(* IEC 61131-3 sources: programs/VI-54/VI-54_20171205/VI-54_20171205/Stations/PLC_VI54/VI-54_171014/Class/_VaranDriveBase (part 2) *)

		s_DataObjectA1.p_Handle^.ucCtrlStat := VARAN_DO_SINGLE_RUN;
	end_if;

	//is Axis 2 in use
	if ( ud_Axis.2 ) then
		s_Axis2Data.e_AxisState := _NoInit;
	else
		s_Axis2Data.e_AxisState := _NotUsed;
//		Axis2_Enable.write( 0 );
//		Axis2_ControlWord.DriveEnable := FALSE;

//		s_Axis2Data.s_WriteValues.a_SyncValues[ 0 ] := ( ( Axis2_ControlWord$DINT shl 16 ) or ( Axis2_SetCurrent and 16#FFFF ) )$DINT;
		s_DataObjectA2.p_DataWrite^.sd_Value1 := s_Axis2Data.s_WriteValues.a_SyncValues[ 0 ];

		s_DataObjectA2.p_Handle^.ucCtrlStat := VARAN_DO_SINGLE_RUN;
	end_if;

	//is Axis 3 in use
	if ( ud_Axis.3 ) then
		s_Axis3Data.e_AxisState := _NoInit;
	else
		s_Axis3Data.e_AxisState := _NotUsed;
//		Axis3_Enable.write( 0 );
//		Axis3_ControlWord.DriveEnable := FALSE;

//		s_Axis3Data.s_WriteValues.a_SyncValues[ 0 ] := ( ( Axis3_ControlWord$DINT shl 16 ) or ( Axis3_SetCurrent and 16#FFFF ) )$DINT;
		s_DataObjectA3.p_DataWrite^.sd_Value1 := s_Axis3Data.s_WriteValues.a_SyncValues[ 0 ];

		s_DataObjectA3.p_Handle^.ucCtrlStat := VARAN_DO_SINGLE_RUN;
	end_if;
*)

(*
	b_InitOk := TRUE;

	InitDrive();
*)
END_FUNCTION

FUNCTION VIRTUAL GLOBAL _VaranDriveBase::State::NewInst
	VAR_INPUT
		pPara 	: ^CmdStruct;
		pResult 	: ^results;
	END_VAR
	VAR_OUTPUT
		ret_code 	: iprStates;
	END_VAR
  VAR
  	pStr_HWTRequested : ^CHAR;
    us_HWTRequestedCurrIndex : USINT;
  END_VAR

  pStr_HWTRequested := NIL;
  us_HWTRequestedCurrIndex := 0;

  ret_code:= READY;

	case ( pPara^.uiCmd ) of
		0 : SetAxisOn( pPara^.aPara[ 0 ]$BDINT );

    1 : // list with parameternumbers to skip

        // check if index in range (0-7)
        //if (pPara^.aPara[2] >= 0) & (pPara^.aPara[2] <= (AxisAvailableNo-1)) then
        if (pPara^.aPara[2] < DIASDRIVE_MAX_AXIS) & (aAxisData[pPara^.aPara[2]].e_AxisState <> _NotUsed) then
          s_SkipParameter[pPara^.aPara[2]].us_No    := to_usint(pPara^.aPara[1]); // number of values in memory
          s_SkipParameter[pPara^.aPara[2]].p_Values := (pPara^.aPara[0])$^USINT; // pointer on memory
        end_if;

    CMD_GET_HARDWARE_DIAGNOSIS :

        ret_code := ERROR;
        pStr_HWTRequested := pPara^.aPara[0]$t_HWCGetHardwareTreeEntryIn.pStr_LastHardewareTreeEntry;

        if pStr_HWTRequested & p_ObjectPath then
          // Needed as default for
          ret_code := READY;

          if (pStr_HWTRequested$^USINT^ = p_ObjectPath^) then // Check if the call was to the Mng
            // Call base 1st as it as info from SPI accesses
            ret_code := Varan_Base::State.NewInst(pPara, pResult);  // Pass on command to base
          end_if;

          if (p_DriveMngBase) then

            // Call Mng, may overwrite some data, has got at least additional info on the FW version
            ret_code := p_DriveMngBase$^VirtualBase^.NewInst(pPara,pResult);

          end_if;
        end_if;

    CMD_GET_HARDWARE_TREE_ENTRY :

        ret_code := ERROR;

        pStr_HWTRequested := pPara^.aPara[0]$t_HWCGetHardwareTreeEntryIn.pStr_LastHardewareTreeEntry;

        // Check HWT String
        if pStr_HWTRequested & p_ObjectPath then

          // Check if the passed string is smaller than the own string
          if pStr_HWTRequested$^USINT^ < p_ObjectPath^ then

            // Call base
            ret_code := Varan_Base::State.NewInst(pPara, pResult);  // Pass on command to base

          // Check if last call was to Base itself
          // Compare string content
          elsif _memcmp( ptr1 := pStr_HWTRequested + 2,
                         ptr2 := p_ObjectPath + 1,
                         cntr := p_ObjectPath^) = 0 then

            // Compare string length
            if (pStr_HWTRequested$^USINT^ = p_ObjectPath^) then

              // Last module called was the Drivemng itself, next module is the 1st axis behind the manager
              if (p_DriveMngBase) then

                ret_code := p_DriveMngBase$^VirtualBase^.NewInst(pPara, pResult); // Pass on command to drive manager

              end_if;

            elsif (pStr_HWTRequested$^USINT^ > p_ObjectPath^ + 1) then // Must be at least 2 Bytey larger, ESCAPE Sequence + Place

              // Check escape sequence
              if ( (pStr_HWTRequested + (p_ObjectPath^) + 2 )^ = HWT_ESCAPE_DRIVE) then // First place after manager Itself is escape sequence + 1 for addional length byte
                // Last Module must have been a Axis Module behind the manager
                // Update index
                pPara^.aPara[0]$t_HWCGetHardwareTreeEntryIn.us_current_index  := p_ObjectPath^ + 3; // Second place after manager Itself is place + 1 for addional length byte
                pPara^.aPara[0]$t_HWCGetHardwareTreeEntryIn.us_current_length := pStr_HWTRequested^ - p_ObjectPath^ - 1;

                if (p_DriveMngBase) then

                  ret_code := p_DriveMngBase$^VirtualBase^.NewInst(pPara, pResult); // Pass on command to drive manager

                end_if;

              else // Length not equal and no Escape sequence, = VARAN Module behind CTMS was called 1.st

                ret_code := Varan_Base::State.NewInst(pPara, pResult);  // Pass on command to base
              end_if;

            else  // Requested string length > this string length, _memcmp failed => Last string was from a differet Varan Port

              ret_code := Varan_Base::State.NewInst(pPara, pResult);  // Pass on command to base
            end_if;

          else
            ret_code := Varan_Base::State.NewInst(pPara, pResult);  // Pass on command to base
          end_if;

        else
          // pStr_HWTRequested is probably nil, pass on command to base
          ret_code := Varan_Base::State.NewInst(pPara, pResult);  // Pass on command to base
        end_if;

	  else
      //Pass on command to base
      ret_code := Varan_Base::State.NewInst(pPara:=pPara, pResult:=pResult);
	end_case;

END_FUNCTION

FUNCTION _VaranDriveBase::SkipEntries
	VAR_INPUT
		us_Axis 	: USINT;
		p_Axis 	: ^t_AxisData;
	END_VAR
  VAR
  	i         : UDINT;
    p_ActPara : ^USINT;
    b_ParaOK  : BOOL;
  END_VAR

  // if there are parameters to skip
  if s_SkipParameter[us_Axis].us_No > 0 then
    b_ParaOK := FALSE;

    // as long as the parameter is skipped and we have have still parameters in the list
    while (b_ParaOK = FALSE) & (p_Axis^.ui_ParaListCnt) do
      // set pointer on first value to skip
      p_ActPara := s_SkipParameter[us_Axis].p_Values;

      b_ParaOK := TRUE;

      // for all skip parameters
      for i := 0 to (s_SkipParameter[us_Axis].us_No - 1) do
        // if the actual parameter number is found in the skip parameter list
        if p_ActPara^ = p_Axis^.p_ParaList^.us_number then
          p_Axis^.ui_ParaListCnt 	-= 1;
          p_Axis^.p_ParaList 		  += sizeof( t_ParaList );

          b_ParaOK := FALSE;
          exit;
        end_if;

        p_ActPara += sizeof(USINT);
      end_for;
    end_while;
  end_if;

END_FUNCTION

FUNCTION GLOBAL _VaranDriveBase::StartCommunication
	VAR_INPUT
		AxisExtend 	: BDINT;
		AxisFast 	: BDINT;
		pServer4CallBack 	: ^BDINT;
	END_VAR

  ExtendedAxisSettings := AxisExtend;
  FastAxisSettings := AxisFast;

  pCallBackServer := pServer4CallBack - sizeof(SvrCh.pMeth);

END_FUNCTION

FUNCTION GLOBAL _VaranDriveBase::GetAxisRdPtr
	VAR_INPUT
		AxisNr 	: DINT;
	END_VAR
	VAR_OUTPUT
		pReadPara 	: ^t_ReadValuePtr;
	END_VAR

  pReadPara := NIL;

  //look which Axis we have
//  if (AxisNr >= 0) & (AxisNr <= (AxisAvailableNo-1)) then
  if (AxisNr < DIASDRIVE_MAX_AXIS) & (aAxisData[AxisNr].e_AxisState <> _NotUsed) then
    pReadPara := #aAxisData[AxisNr].s_ReadValues;
  end_if;

END_FUNCTION

FUNCTION GLOBAL _VaranDriveBase::GetAxisWrPtr
	VAR_INPUT
		AxisNr 	: DINT;
	END_VAR
	VAR_OUTPUT
		pWritePara 	: ^t_WriteValuePtr;
	END_VAR

  pWritePara := NIL;

  //look which Axis we have
//  if (AxisNr >= 0) & (AxisNr <= (AxisAvailableNo-1)) then
  if (AxisNr < DIASDRIVE_MAX_AXIS) & (aAxisData[AxisNr].e_AxisState <> _NotUsed) then
    pWritePara := #aAxisData[AxisNr].s_WriteValues;
  end_if;

END_FUNCTION

FUNCTION GLOBAL _VaranDriveBase::GetDriveIntState
	VAR_OUTPUT
		retcode 	: DINT;
	END_VAR

  // to get the actual state of the rtwork state machine
  // retcode = 3 means Operational (MOD 4 is for model SDD100/5000 to have the same returncodes)
  retcode := e_RtSSW$DINT MOD 4;

END_FUNCTION

FUNCTION _VaranDriveBase::GetObjectValueNew
	VAR_INPUT
		us_Axis 	: USINT;
	END_VAR
  VAR
    p_Axis			: ^t_AxisData;
    p_Write     : ^t_newASYWrite;
    p_Read      : ^t_newASYRead;
  END_VAR

	//------------------------------------------------------------------------------------------------
	//look which Axis we have and set pointers
//  if (us_Axis >= 0) & (us_Axis <= (AxisAvailableNo-1)) then
  if (us_Axis < DIASDRIVE_MAX_AXIS) & (aAxisData[us_Axis].e_AxisState <> _NotUsed) then
    p_Axis	:= #aAxisData[us_Axis];
    p_Read 	:= newAsyDO.p_DataRead + us_Axis * sizeof(t_newASYRead);
    p_Write	:= newAsyDO.p_DataWrite + us_Axis * sizeof(t_newASYWrite);
  else
    //else do nothing (should not come her)
    return;
  end_if;

	//------------------------------------------------------------------------------------------------
	//get to right step
	case ( p_Axis^.us_ParaReady ) of

		_SendExecution: // we wait 1 cycle to ensure that the request is written to the Drive (what object number we want to read or write)
							p_Axis^.us_ParaReady := _ResetExecution;

    _ResetExecution:// now toggle the togglebit to start tell the drive, that the data are complete (no chance for byte errors in this way)

              //send transmit execution request for object handling
							p_Axis^.b_OldToggleState := p_Read^.us_TransmitControl.ToggleBit;

              // toggle toggle bit
              p_Write^.us_DriveControl.ToggleBit := NOT p_Read^.us_TransmitControl.ToggleBit;

							//reset error and go to next step
							p_Axis^.sd_ObjectError := 0;
							p_Axis^.us_ParaReady := _Wait4Response;

		_Wait4Response:		//wait until receive state is true
							if ( p_Read^.us_TransmitControl.ToggleBit <> p_Axis^.b_OldToggleState) then

								//look if we have a parameter list
								if ( p_Axis^.b_ListActive = TRUE ) then

                  // skip all defined parameter entries
                  SkipEntries(us_Axis, p_Axis);

									//have we set all parameter
									if ( p_Axis^.ui_ParaListCnt ) then

										//set data to object handling registers
										p_Write^.us_ObjectAddress					        := p_Axis^.p_ParaList^.us_number;
										p_Write^.sd_ObjectValue					          := p_Axis^.p_ParaList^.sd_value;
										p_Write^.us_DriveControl.ReadWriteObject	:= TRUE;

										//set next parameter step and set pointer to next parameter data
										p_Axis^.us_ParaReady 	:= _SendExecution;
										p_Axis^.ui_ParaListCnt 	-= 1;
										p_Axis^.p_ParaList 		+= sizeof( t_ParaList );

									else
										//set ssw to idle and deactivate parameter list
										p_Axis^.b_ListActive 	:= FALSE;

										//look if we get a parameter list
										if ( p_Axis^.e_AxisState = _NoParaList ) then
											p_Axis^.e_AxisState		:= _NotSynchron;
										end_if;

										p_Axis^.us_ParaReady 	:= _IdleState;

									end_if;

								else
									//get to idle step
									p_Axis^.us_ParaReady := _IdleState;

									//look for an object error
									if ( p_Read^.us_TransmitControl.ErrorInObjectHandling = TRUE ) then
										p_Axis^.sd_ObjectError := p_Read^.sd_ObjectValue;
									else
                 		p_Axis^.sd_Asyncdata := p_Read^.sd_ObjectValue;
                  end_if;

								end_if;
							end_if;

		_IdleState:				//do nothing in this step

	end_case;

END_FUNCTION

FUNCTION _VaranDriveBase::InitAxisNew
	VAR_INPUT
		us_AxisNo 	: USINT;
	END_VAR
	VAR_OUTPUT
		sd_retval 	: DINT;
	END_VAR
  VAR
    p_Axis			: ^t_AxisData;
    p_Write     : ^t_newASYWrite;
    p_Read      : ^t_newASYRead;
    p_data_object : ^t_newISODO;
  END_VAR

	//we do this only if class is not initialized
	if ( State <> _NotInitialized ) then
		return;
	end_if;

	//------------------------------------------------------------------------------------------------
	//look which Axis we have and set pointers
//  if (us_AxisNo >= 0) & (us_AxisNo <= (AxisAvailableNo-1)) then
  if (us_AxisNo < DIASDRIVE_MAX_AXIS) & (aAxisData[us_AxisNo].e_AxisState <> _NotUsed) then
    p_Axis			:= #aAxisData[us_AxisNo];
    p_data_object	:= #newIsoDOs[us_AxisNo];
    p_Read 	:= newAsyDO.p_DataRead + us_AxisNo * sizeof(t_newASYRead);
    p_Write	:= newAsyDO.p_DataWrite + us_AxisNo * sizeof(t_newASYWrite);
  else
    sd_retval := -2;
    return;
  end_if;

	//------------------------------------------------------------------------------------------------
	//look which case we have
	case ( e_InitSSW ) of

		//-----------------------------------------------------------------------------------------------
		_SetDataObjectOn:
					//is Axis in use
					if ( p_Axis^.e_AxisState <> _NotUsed ) then

//Revision 1.20 start
            _memset(p_data_object^.p_DataWrite, 16#00, p_Axis^.ud_DOLength); // reinit the memory before sending
//Revision 1.20 end

						//reset data object of Axis
            if b_PayloadSupport then
              if bAddDOsToListSupport then
                sd_retval := MULTI_VARAN_IINSERTDOINTODOL(p_data_object^.p_Handle$UDINT);
              end_if;
              EnableDO(ud_DOHandle:=p_data_object^.p_Handle$UDINT);
            else
                // Payload DOs automatically use the client Timebase to set the Prescaler of the DOs
              //set right multiplier
              p_data_object^.p_Handle^.ucExePrescaler := VaranTimeMultiplier$USINT - 1;

              ResetDataObject	( p_handleDO	:= p_data_object^.p_Handle
                              , us_state		:= VARAN_DO_CONT_RUN
                                , ud_bytes		:= p_Axis^.ud_DOLength * 2);
            end_if;
(*
            if ( us_AxisNo = 3 & UseFastAxis ) then

              ResetDataObject	( p_handleDO	:= s_DataFastAxis.p_Handle
                              , us_state		:= VARAN_DO_CONT_RUN
                              , ud_bytes		:= sizeof( t_FastAxisRead ) + sizeof( t_FastAxisWrite )
                              );

              s_DataFastAxis.p_DataWrite^.us_TransmittExecution.EnableType2 := TRUE;
            end_if;
*)
						//next step
						e_InitSSW := _SetInitAxis;

					else
						//go to idle state
						e_InitSSW := _CyIdle;
					end_if;

		//-----------------------------------------------------------------------------------------------
		_SetInitAxis:
					//InitAxis
					if ( p_Axis^.e_AxisState = _NoInit ) then

						p_Write^.us_DriveControl.InitCommunication 			:= TRUE;

					end_if;

          p_Axis^.b_OldToggleState := p_Read^.us_TransmitControl.ToggleBit;

          // toggle toggle bit
          p_Write^.us_DriveControl.ToggleBit := NOT p_Read^.us_TransmitControl.ToggleBit;

					//next step and timestamp
					e_InitSSW 		:= _WaitInit;
					ud_TimemarkInit := ops.tAbsolute;

		//-----------------------------------------------------------------------------------------------
		_WaitInit:	//reset startobjecttransfer bit

					//look if Axis 1 must be init
					if ( p_Axis^.e_AxisState = _NoInit ) then

						//object must be executed, error in object handling must be set and error code must be 9
						if (( p_Read^.us_TransmitControl.ToggleBit <> p_Axis^.b_OldToggleState)
                & p_Read^.us_TransmitControl.ErrorInObjectHandling	= TRUE
                & p_Read^.sd_ObjectValue 							= 9
                )
						then
							//set Axis to next state
							p_Axis^.e_AxisState := _NoParaList;
							e_InitSSW := _SetFinishInit;

            //after timeout check again
            elsif ( ops.tAbsolute - ud_TimemarkInit > 1sec ) then
              e_InitSSW := _SetInitAxis;
            end_if;

					//after timeout check again
					elsif ( ops.tAbsolute - ud_TimemarkInit > 1sec ) then
						e_InitSSW := _SetInitAxis;
					end_if;

		//-----------------------------------------------------------------------------------------------
		_SetFinishInit:

					//If Axis is in right state
					if ( p_Axis^.e_AxisState = _NoParaList ) then

						p_Write^.us_DriveControl.InitCommunication 			:= FALSE;
					end_if;

          p_Axis^.b_OldToggleState := p_Read^.us_TransmitControl.ToggleBit;

          // toggle toggle bit
          p_Write^.us_DriveControl.ToggleBit := NOT p_Read^.us_TransmitControl.ToggleBit;

					//next step and timestamp
					e_InitSSW 		:= _GetFinishInit;
					ud_TimemarkInit := ops.tAbsolute;

		//-----------------------------------------------------------------------------------------------
		_GetFinishInit:

					//look if Axis is in use and error bit is reset
					if	( p_Read^.us_TransmitControl.ErrorInObjectHandling = FALSE) &
						  ( p_Read^.us_TransmitControl.ToggleBit <> p_Axis^.b_OldToggleState)
					then
					//reset startobjecttransfer bit

						//final step, init ok and class ok
						e_InitSSW := _CyIdle;

					else

						//try again if return value is 10 or 8 (see DiasDrive Doku)
						if	( ( p_Read^.sd_ObjectValue = 10 | p_Read^.sd_ObjectValue = 8 )
							& p_Read^.us_TransmitControl.ErrorInObjectHandling = TRUE
							)
						then
							e_InitSSW 			:= _SetInitAxis;
							p_Axis^.e_AxisState := _NoInit;
						end_if;

						//if timeout check again
						if ( ops.tAbsolute - ud_TimemarkInit > 2sec ) then
							e_InitSSW := _SetFinishInit;
						end_if;
					end_if;

		//-----------------------------------------------------------------------------------------------
		_CyIdle:

	end_case;

	//return ssw
	sd_retval := e_InitSSW$DINT;

END_FUNCTION

FUNCTION GLOBAL _VaranDriveBase::ExternInitFinished

  // if all axis parameters have been sent
  if b_CompatibilityMode then
    e_RtSSW := CompWaitForSynchrony;
  else
    e_RtSSW := WaitForSynchrony;
  end_if;

END_FUNCTION

FUNCTION _VaranDriveBase::GetDriveType
	VAR_INPUT
		HWCode 	: DINT;
	END_VAR
  VAR_OUTPUT
    AxisNo  : SINT;
  END_VAR
  VAR
  	DriveType : DINT;
  END_VAR

  DriveType := HWCode SHR 16;

  case DriveType of

  // 3 Axis **************************************************************************
    0..4, 6, 12, 16, 20, 26:
      AxisNo := 3;
      AxisAvailableHW := 2#111;

  // 2 Axis **************************************************************************
    5, 9:// SDD215 and SDD210 special case
      AxisNo := 3; // we need to simulate 3 axis, because of the skipped axis
      AxisAvailableHW := 2#101;
      if ExtendedAxisSettings.2 = TRUE then
        ExtendedAxisSettings.2 := FALSE;
        ExtendedAxisSettings.3 := TRUE;
      end_if;
      if FastAxisSettings.2 = TRUE then
        FastAxisSettings.2 := FALSE;
        FastAxisSettings.3 := TRUE;
      end_if;

      b_IsSDD21x := TRUE;

    22:// SDD205 normal case
      AxisNo := 2;
      AxisAvailableHW := 2#11;

  // 1 Axis **************************************************************************
    7, 21, 10:
      AxisNo := 1;
      AxisAvailableHW := 2#1;
  else
    AxisNo := -1;
  end_case;

END_FUNCTION

FUNCTION VIRTUAL GLOBAL _VaranDriveBase::UpdateRtPostScan
  VAR
    i           : UDINT;
  END_VAR

//=================================================================================================
#ifdef VM_CLASS_TIME_MEASUREMENT
	StartTimeMeasurement(VARANTIME_RTPOSTSCAN);
#endif
//=================================================================================================

  IF Online & b_CompatibilityMode & AxisAvailableNo THEN
    FOR i := 0 TO (AxisAvailableNo-1) DO
      IF aDataObjects[i].b_NewAsyDataTemp & aDataObjects[i].p_DataWrite THEN
        aAxisData[i].us_ParaReady := _SendExecution;

//        _memcpy(  ptr1:= aDataObjects[i].p_DataWrite
//                , ptr2:= #aDataObjects[i].AsyDataTemp
//                , cntr:= aAxisData[i].ud_DOLength
//                );
        aDataObjects[i].p_DataWrite^.us_ObjectAddress := aDataObjects[i].AsyDataTemp.us_ObjectAddress;
        aDataObjects[i].p_DataWrite^.sd_ObjectValue := aDataObjects[i].AsyDataTemp.sd_ObjectValue;
        aDataObjects[i].p_DataWrite^.us_DriveControl.ReadWriteObject := aDataObjects[i].AsyDataTemp.us_DriveControl.ReadWriteObject;

        // aDataObjects[i].p_DataWrite^ := aDataObjects[i].AsyDataTemp;

        aDataObjects[i].b_NewAsyDataTemp := FALSE;
        EXIT;
      END_IF;
    END_FOR;
  END_IF;

  if b_UpdateThisTime then

    if Online then
      case e_RtSSW of

        // Comp = compatibility mode to dias drive 300 series

        // ******************************************************************************************************************************************

        CompOperational:

          if AxisAvailableNo then
            for i := 0 to (AxisAvailableNo-1) do
              if ( aAxisData[i].e_AxisState <> _NotUsed ) then
                if aAxisData[i].b_ExtendedAxis then
                  _memcpy(#aDataObjects[i].p_DataWrite^.sd_Value1, #aAxisData[i].s_WriteValues.a_SyncValues[ 0 ], 5 * sizeof(DINT));
                else
                  aDataObjects[i].p_DataWrite^.sd_Value1 := aAxisData[i].s_WriteValues.a_SyncValues[ 0 ];
                  aDataObjects[i].p_DataWrite^.sd_Value2 := aAxisData[i].s_WriteValues.a_SyncValues[ 1 ];
                end_if;
              end_if;
            end_for;
          end_if;

        // ******************************************************************************************************************************************
        // now the part for DiasDrive 100/5000 series

        Operational:

          if AxisAvailableNo then
            for i := 0 to (AxisAvailableNo-1) do
              if ( aAxisData[i].e_AxisState <> _NotUsed ) then
                if aAxisData[i].b_ExtendedAxis then
                  _memcpy(#newIsoDOs[i].p_DataWrite^.Value1, #aAxisData[i].s_WriteValues.a_SyncValues[ 0 ], sizeof(t_newReadDataOneAxis));
                else
                  newIsoDOs[i].p_DataWrite^.Value1 := aAxisData[i].s_WriteValues.a_SyncValues[ 0 ];
                  newIsoDOs[i].p_DataWrite^.Value2 := aAxisData[i].s_WriteValues.a_SyncValues[ 1 ];
                end_if;
              end_if;
            end_for;
          end_if;

      end_case;
    end_if;
  end_if;

//=================================================================================================
#ifdef VM_CLASS_TIME_MEASUREMENT
	StopTimeMeasurement(VARANTIME_RTPOSTSCAN);
#endif
//=================================================================================================

END_FUNCTION

FUNCTION GLOBAL _VaranDriveBase::GetSeries
	VAR_OUTPUT
		retcode 	: USINT;
	END_VAR

  if b_CompatibilityMode = TRUE then
    retcode := 0;
  else
    retcode := 1;
  end_if;

END_FUNCTION

FUNCTION GLOBAL _VaranDriveBase::IsSDD21x
	VAR_OUTPUT
		retcode 	: BOOL;
	END_VAR

  retcode := b_IsSDD21x;

END_FUNCTION

FUNCTION VIRTUAL GLOBAL _VaranDriveBase::CheckDeviceID
	VAR_INPUT
		ID2Check 	: UDINT;
	END_VAR
	VAR_OUTPUT
		IsOK 	: BOOL;
	END_VAR

	//look if it is right hardware
	if ((ID2Check <> VAC011_DEVICE_ID )
	&   (ID2Check <> VAC012_DEVICE_ID )
	&   (ID2Check <> VAC013_DEVICE_ID )
  &   (ID2Check <> DIASDRIVE_MINI_DEVICE_ID )
  &   (ID2Check <> DIASDRIVE_MAXI_DEVICE_ID )) then
		IsOK := FALSE;
  else
    IsOK := TRUE;
  end_if;

END_FUNCTION

FUNCTION VIRTUAL GLOBAL _VaranDriveBase::UpdateCy
VAR
	i : UDINT;
  sd_retval : DINT;
END_VAR

//=================================================================================================
#ifdef VM_CLASS_TIME_MEASUREMENT
	StartTimeMeasurement(VARANTIME_CY);
#endif
//=================================================================================================

  IF Online THEN
    IF b_CompatibilityMode = FALSE then
      if AxisAvailableNo THEN
        CASE e_RtSSW OF
          // ******************************************************************************************************************************************
          InitAxis, GetSendParaList, Operational, WaitForSynchrony:
            FOR i := 0 TO (AxisAvailableNo-1) DO
              IF newAsyDO.b_NewAsyDataTemp[i] & newAsyDO.p_DataWrite THEN
                aAxisData[i].us_ParaReady := _SendExecution;
                newAsyDO.p_DataWrite^[i] := newAsyDO.AsyDataTemp[i];
                newAsyDO.b_NewAsyDataTemp[i] := FALSE;
                EXIT;
              END_IF;
            END_FOR;
        END_CASE;
      end_if;

      case e_RtSSW of
        // ******************************************************************************************************************************************
        // now the part for DiasDrive 100/5000 series
        // ******************************************************************************************************************************************
        // ******************************************************************************************************************************************
        InitAxis:
          if bAddDOsToListSupport then
            AddIsoDOsNew();
          end_if;

          // ******************************************************************************************************************************************
          // enable sync of varan and drive for DiasDrive 100/5000 series
          // ******************************************************************************************************************************************
          if ( b_SyncEnabled = FALSE)
          & AxisAvailableNo then
            if CreatedNewAsyDOs = FALSE then
              if b_PayloadSupport then
                sd_retval := AddRdWrPayloadDO(  ud_dol_type     :=  VARAN_DOL_ASY
                                              , p_ud_handle     := ( #newAsyDO.p_Handle )$^UDINT
                                              , ud_offset_read  :=  DIASDRIVE_ADR_SERVICE + DIASDRIVE_ADR_SERVICE_READ
                                              , ud_length_read  := AxisAvailableNo * sizeof(t_newASYRead)
                                              , p_ud_data_read  := ( #newAsyDO.p_DataRead )$^UDINT
                                              , ud_offset_write := DIASDRIVE_ADR_SERVICE + DIASDRIVE_ADR_SERVICE_WRITE
                                              , ud_length_write := AxisAvailableNo * sizeof(t_newASYWrite)
                                              , p_ud_data_write := ( #newAsyDO.p_DataWrite )$^UDINT
                                              , ud_type         := VM_MEMORY_ACCESS);

                //look if an error occurs
                if ( sd_retval <> VARANMANAGER_OK ) then
                  State := _CreateDOFailed;
                  return;
                end_if;
              else
                // create 1 general ASY RdWrDO with variable size (depending on number of available axis)
                sd_retval := VaranIn.AddRdWrDO	( p_us_position_info:= p_VaranPosition
                                , ud_dol_type		:= VARAN_DOL_ASY
                                , p_ud_handle		:= ( #newAsyDO.p_Handle )$^UDINT
                                , ud_address_read	:= 0
                                , ud_length_read	:= AxisAvailableNo * sizeof(t_newASYRead)
                                , p_ud_data_read	:= ( #newAsyDO.p_DataRead )$^UDINT
                                , ud_address_write	:= 0
                                , ud_length_write	:= AxisAvailableNo * sizeof(t_newASYWrite)
                                , p_ud_data_write	:= ( #newAsyDO.p_DataWrite )$^UDINT
                                , ud_type			:= VM_MEMORY_ACCESS
                                );

                //look if an error occurs
                if ( sd_retval <> VARANMANAGER_OK ) then
                  State := _CreateDOFailed;
                  return;
                end_if;

                //get address pointer to change address of access
                newAsyDO.p_DOSettings := (newAsyDO.p_DataWrite)$^t_VaranDOSettingsRdWr - VM_DO_OFFSET_RDWR;
              end_if;
              CreatedNewAsyDOs := TRUE;
            end_if;

            if b_PayloadSupport then
              EnableDO(ud_DOHandle:=newAsyDO.p_Handle$UDINT);
            else
              //correct access address
              newAsyDO.p_DOSettings^.ud_AddressRd := DeviceAddress + DIASDRIVE_ADR_SERVICE + DIASDRIVE_ADR_SERVICE_READ;
              newAsyDO.p_DOSettings^.ud_AddressWr := DeviceAddress + DIASDRIVE_ADR_SERVICE + DIASDRIVE_ADR_SERVICE_WRITE;

              //reset data object of Axis
              ResetDataObject	( p_handleDO	:= newAsyDO.p_Handle
                              , us_state		:= VARAN_DO_CONT_RUN
                              , ud_bytes		:= AxisAvailableNo * sizeof(t_newASYRead) + AxisAvailableNo * sizeof(t_newASYWrite)
                              );
            end_if;

            sd_retval := EnableSyncOut	( us_sync_nr				:= 0
                                        , sd_offset					:= sd_SyncOffset
                                        , us_period_multiplier		:= VaranTimeMultiplier$USINT
                                        , us_frame_count_treshold	:= 0
                                        , us_enable_frame_count		:= 0
                                        , b_use_divider_sync := FALSE
                                        );

            //look for an error
            if ( sd_retval <> VARANMANAGER_OK ) then
              return;
            end_if;

            sd_retval := EnableSyncOut	( us_sync_nr				:= 1
                                        , sd_offset					:= sd_SyncOffset MOD 6250
                                        , us_period_multiplier		:= 0
                                        , us_frame_count_treshold	:= 0
                                        , us_enable_frame_count		:= 0
                                        , b_use_divider_sync := TRUE
                                        );

            //look for an error
            if ( sd_retval <> VARANMANAGER_OK ) then
              return;
            end_if;

            b_SyncEnabled := TRUE;
            return;
          end_if;

          //switch Axis
          if e_InitSSW <> _SetDataObjectOn then
            case ( us_AxisNumber ) of

              1..DIASDRIVE_MAX_AXIS: 	//wait until Axis are initialized
                if us_AxisNumber <= AxisAvailableNo then
                  if InitAxisNew( us_AxisNo := us_AxisNumber-1 ) = _CyIdle$DINT then
                    us_AxisNumber 	+=1;
                    e_InitSSW 	:= _SetDataObjectOn;
                  end_if;
                else
                  us_AxisNumber := DIASDRIVE_MAX_AXIS+1;
                end_if;
            end_case;
          end_if;

        // ******************************************************************************************************************************************
        GetSendParaList, Operational:
          // update asynchron parameters
          if AxisAvailableNo then
            for i := 0 to (AxisAvailableNo-1) do
              //Axis "i" object value
              GetObjectValueNew( us_Axis := to_usint(i) );
            end_for;
          end_if;
      end_case;

    ELSE  //b_CompatibilityMode = TRUE
      case e_RtSSW of
        //*****************************************************************************
        //**      Comp = compatibility mode to dias drive 300 series                 **
        //*****************************************************************************
        CompInitAxis:

          if bAddDOsToListSupport then
            InstallDefaultDO();
          end_if;

          if b_AlreadyConnected = TRUE then

            //*****************************************************************************
            //**  switch Axis                                                            **
            //*****************************************************************************
            case ( us_AxisNumber ) of

              // ***********************************************************************************************************************************
              0:	//is done at rt task

              // ***********************************************************************************************************************************
              1: 	//wait until first axis is initialized
              // must be done at realtime task

              // ***********************************************************************************************************************************
              2: // we check how many axis are really available (parameter communication)
                case GetCompAxisSSW of
                  // ***********************************************************************************************************************************
                  0: //is done at rt-task

                  // ***********************************************************************************************************************************
                  1: //is done at rt-task

                  // ***********************************************************************************************************************************
                  2:
                    //Check if we can use the new interface and add DOs in UpdateCy
                    if bAddDOsToListSupport then
                      //Do nothing, DOs are installed in UpdateCy
                      //We have the old interface, install DOs here
                      AddIsoDOsCompMode();
                    end_if;

                end_case;
            end_case;
          end_if;
      end_case;
    END_IF;
  END_IF;

//=================================================================================================
#ifdef VM_CLASS_TIME_MEASUREMENT
	StopTimeMeasurement(VARANTIME_CY);
#endif
//=================================================================================================

END_FUNCTION

FUNCTION GLOBAL _VaranDriveBase::SetObjectCallBack
	VAR_INPUT
		p_DriveMngBaseNew 	: ^void;
	END_VAR

  p_DriveMngBase := p_DriveMngBaseNew;

END_FUNCTION

FUNCTION _VaranDriveBase::AddIsoDOsCompMode
VAR
	i : UDINT;
  sd_retval : DINT;
  tmp_dol_Type: UDINT;
END_VAR

  // if we got more than 1 axis and the last axis has no VARAN handle yet
  if (AxisAvailableNo > 1) & (DataInitFinished = FALSE) then
    if (aDataObjects[AxisAvailableNo-1].p_Handle = NIL) then

      for i := 1 to AxisAvailableNo-1 do

        if AxisAvailableHW AND (1 SHL i$UDINT) then

          //set right data object length
          if (1 SHL i$UDINT) AND ExtendedAxisSettings then
            aAxisData[i].ud_DOLength := sizeof(t_DataReadOneAxis);
            aAxisData[i].b_ExtendedAxis := TRUE;
          else
            aAxisData[i].ud_DOLength := sizeof(t_DataReadOneAxis) - 3 * sizeof(DINT);
            aAxisData[i].b_ExtendedAxis := FALSE;
          end_if;

          // check for fastaxis
          if (1 SHL i$UDINT) AND FastAxisSettings then
            aAxisData[i].b_FastAxis := TRUE;
          else
            aAxisData[i].b_FastAxis := FALSE;
          end_if;

          //install data object
          if b_PayloadSupport then

            tmp_dol_type := VARAN_DOL_ISO;

            if bAddDOsToListSupport then
              tmp_dol_Type := tmp_dol_Type OR VARAN_DOL_NOT_INSERT_DO_INTO_DOL;
            end_if;

            sd_retval := AddRdWrPayloadDO(  ud_dol_type     := tmp_dol_type
                                          , p_ud_handle     := ( #aDataObjects[ i ].p_Handle )$^UDINT
                                          , ud_offset_read  := i$UDINT*DIASDRIVE_OFFSET_Axis + DIASDRIVE_OFFSET_AxisRead
                                          , ud_length_read  := aAxisData[i].ud_DOLength
                                          , p_ud_data_read  := ( #aDataObjects[ i ].p_DataRead )$^UDINT
                                          , ud_offset_write := i$UDINT*DIASDRIVE_OFFSET_Axis
                                          , ud_length_write := aAxisData[i].ud_DOLength
                                          , p_ud_data_write := ( #aDataObjects[ i ].p_DataWrite )$^UDINT
                                          , ud_type         := VM_MEMORY_ACCESS);

            //look if an error occurs
            if ( sd_retval <> VARANMANAGER_OK ) then
              State := _CreateDOFailed;
              return;
            end_if;
          else
            sd_retval := VaranIn.AddRdWrDO	( p_us_position_info:= p_VaranPosition
                            , ud_dol_type		:= VARAN_DOL_ISO
                            , p_ud_handle		:= ( #aDataObjects[i].p_Handle )$^UDINT
                            , ud_address_read	:= 0
                            , ud_length_read	:= aAxisData[i].ud_DOLength
                            , p_ud_data_read	:= ( #aDataObjects[i].p_DataRead )$^UDINT
                            , ud_address_write	:= 0
                            , ud_length_write	:= aAxisData[i].ud_DOLength
                            , p_ud_data_write	:= ( #aDataObjects[i].p_DataWrite )$^UDINT
                            , ud_type			:= VM_MEMORY_ACCESS
                            );

            //look if an error occurs
            if ( sd_retval <> VARANMANAGER_OK ) then
              State := _CreateDOFailed;
              return;
            end_if;

//            //get address pointer to change address later when module is connected
//            aDataObjects[i].p_DOSettings := (aDataObjects[i].p_DataWrite)$^t_VaranDOSettingsRdWr - VM_DO_OFFSET_RDWR;
          end_if;
            //get address pointer to change address later when module is connected
            aDataObjects[i].p_DOSettings := (aDataObjects[i].p_DataWrite)$^t_VaranDOSettingsRdWr - VM_DO_OFFSET_RDWR;

        end_if;
      end_for;
    end_if;

    for i := 1 to AxisAvailableNo-1 do

      if AxisAvailableHW AND (1 SHL i$UDINT) then
        if b_PayloadSupport =FALSE then
        //correct address for data object read/write Axis 1
        aDataObjects[i$UDINT].p_DOSettings^.ud_AddressRd := DeviceAddress + i$UDINT*DIASDRIVE_OFFSET_Axis + DIASDRIVE_OFFSET_AxisRead;
        aDataObjects[i$UDINT].p_DOSettings^.ud_AddressWr := DeviceAddress + i$UDINT*DIASDRIVE_OFFSET_Axis;
        end_if;
        //set enable outputs in DCB
        //with VAC012 the hardware enables the outputs
        if ( DeviceID = VAC011_DEVICE_ID ) then
          aDataObjects[i].p_DataWrite^.us_DriveControl := 2#00111000;
        end_if;

        //set transmit register
        if aAxisData[i$UDINT].b_ExtendedAxis then
          aDataObjects[i$UDINT].p_DataWrite^.us_TransmitExecution.EnableValue3_5 := TRUE;
        end_if;

        //set right para state
        aAxisData[i].us_ParaReady := _IdleState;
        aAxisData[i].e_AxisState := _NoInit;
      end_if;
    end_for;

    DataInitFinished := TRUE;
    GetCompAxisSSW += 1;

  elsif AxisAvailableNo = 1 then
  //For SDD115/120, we have to set DataInitFinished TRUE to leave this if.
  //DataInitFinished will be set in the Method AddIsoDOsCompMode when we have more axis.
    DataInitFinished := TRUE;

  end_if;

END_FUNCTION

FUNCTION _VaranDriveBase::AddIsoDOsNew
VAR
	i : UDINT;
  tmp_dol_type : UDINT;
  sd_retval : DINT;
END_VAR

  if CreatedNewIsoDOs = FALSE then
    AxisAvailableNo := 0;

    // create a ISO RdWr DO for every available axis
    for i := 0 to (DIASDRIVE_MAX_AXIS*DIASDRIVE_MAX_AXIS_PER_MODULE-1) do

      if (1 SHL i$UDINT) AND AxisAvailableHW then

        if (1 SHL i$UDINT) AND ExtendedAxisSettings then
          aAxisData[AxisAvailableNo].ud_DOLength := sizeof(t_newReadDataOneAxis);
          aAxisData[AxisAvailableNo].b_ExtendedAxis := TRUE;
        else
          aAxisData[AxisAvailableNo].ud_DOLength := sizeof(t_newReadDataOneAxis) - 3 * sizeof(DINT);
          aAxisData[AxisAvailableNo].b_ExtendedAxis := FALSE;
        end_if;

        // check for fastaxis
        if (1 SHL i$UDINT) AND FastAxisSettings then
          aAxisData[AxisAvailableNo].b_FastAxis := TRUE;
        else
          aAxisData[AxisAvailableNo].b_FastAxis := FALSE;
        end_if;

        //install data object
        if b_PayloadSupport then

          tmp_dol_type := VARAN_DOL_ISO;

          if bAddDOsToListSupport then
            tmp_dol_Type := tmp_dol_Type OR VARAN_DOL_NOT_INSERT_DO_INTO_DOL;
          end_if;

          sd_retval := AddRdWrPayloadDO(  ud_dol_type     := tmp_dol_type
                                        , p_ud_handle     := ( #newIsoDOs[AxisAvailableNo].p_Handle )$^UDINT
                                        , ud_offset_read  := DIASDRIVE_ADR_ALT_BUF_RD_OFFSET + AxisAvailableNo$UDINT*DIASDRIVE_OFFSET_AxisRead
                                        , ud_length_read  := aAxisData[AxisAvailableNo].ud_DOLength
                                        , p_ud_data_read  := ( #newIsoDOs[AxisAvailableNo].p_DataRead )$^UDINT
                                        , ud_offset_write :=  DIASDRIVE_ADR_ALT_BUF_WR_OFFSET + AxisAvailableNo$UDINT*DIASDRIVE_OFFSET_AxisRead
                                        , ud_length_write := aAxisData[AxisAvailableNo].ud_DOLength
                                        , p_ud_data_write := ( #newIsoDOs[AxisAvailableNo].p_DataWrite )$^UDINT
                                        , ud_type         := VM_MEMORY_ACCESS);

          //look if an error occurs
          if ( sd_retval <> VARANMANAGER_OK ) then
            State := _CreateDOFailed;
            return;
          end_if;
        else
          sd_retval := VaranIn.AddRdWrDO	( p_us_position_info:= p_VaranPosition
                          , ud_dol_type		:= VARAN_DOL_ISO
                          , p_ud_handle		:= ( #newIsoDOs[AxisAvailableNo].p_Handle )$^UDINT
                          , ud_address_read	:= 0
                          , ud_length_read	:= aAxisData[AxisAvailableNo].ud_DOLength
                          , p_ud_data_read	:= ( #newIsoDOs[AxisAvailableNo].p_DataRead )$^UDINT
                          , ud_address_write	:= 0
                          , ud_length_write	:= aAxisData[AxisAvailableNo].ud_DOLength
                          , p_ud_data_write	:= ( #newIsoDOs[AxisAvailableNo].p_DataWrite )$^UDINT
                          , ud_type			:= VM_MEMORY_ACCESS
                          );

          //look if an error occurs
          if ( sd_retval <> VARANMANAGER_OK ) then
            State := _CreateDOFailed;
            return;
          end_if;
        end_if;
        //get address pointer to change address later when module is connected
        newIsoDOs[AxisAvailableNo].p_DOSettings := (newIsoDOs[AxisAvailableNo].p_DataWrite)$^t_VaranDOSettingsRdWr - VM_DO_OFFSET_RDWR;
        AxisAvailableNo += 1;

        if AxisAvailableNo = DIASDRIVE_MAX_AXIS then
          exit;
        end_if;
      end_if;
    end_for;

    // check if we need to get the digital Inputs
    if TempFetchDigitalInputs then
      //install data object
      if b_PayloadSupport then

        tmp_dol_type := VARAN_DOL_ISO;

        if bAddDOsToListSupport then
          tmp_dol_Type := tmp_dol_Type OR VARAN_DOL_NOT_INSERT_DO_INTO_DOL;
        end_if;

        sd_retval := AddRdPayloadDO(  ud_dol_type   := tmp_dol_Type
                                    , p_ud_handle   := ( #newDigInDO.p_Handle)$^UDINT
                                    , ud_offset_read:= DIASDRIVE_ADR_INPUTS
                                    , ud_length_read:= sizeof(USINT)
                                    , p_ud_data_read:= ( #newDigInDO.p_DataRead)$^UDINT
                                    , ud_type       := VM_MEMORY_ACCESS);

        //look if an error occurs
        if ( sd_retval <> VARANMANAGER_OK ) then
          State := _CreateDOFailed;
          return;
        end_if;
      else
        sd_retval := VaranIn.AddRdDO 	( p_us_position_info:= p_VaranPosition
                                      , ud_dol_type	:= VARAN_DOL_ISO
                                      , p_ud_handle	:= ( #newDigInDO.p_Handle )$^UDINT
                                      , ud_address	:= 0
                                      , ud_length	  := sizeof(USINT)
                                      , p_ud_data  	:= ( #newDigInDO.p_DataRead )$^UDINT
                                      , ud_type			:= VM_MEMORY_ACCESS
                                      );

        //look if an error occurs
        if ( sd_retval <> VARANMANAGER_OK ) then
          State := _CreateDOFailed;
          return;
        end_if;

        //get address pointer to change address later when module is connected
        newDigInDO.p_DOSettings := (newDigInDO.p_DataRead)$^t_VaranDOSettingsRd - VM_DO_OFFSET_RD;
      end_if;
    end_if;

    AxisAvailable100 := AxisAvailableNo;
    CreatedNewIsoDOs := TRUE;
  else
    AxisAvailableNo := AxisAvailable100;
  end_if;

  //------------------------------------------------------------------------------------------------
  if b_AlreadyConnected = FALSE & AxisAvailableNo then

    //Init all Axis
    for i := 0 to (AxisAvailableNo-1) do
      // SDD100/5000 model
      if b_PayloadSupport = FALSE then

        //correct address for data object read/write Axis 1
        newIsoDOs[i].p_DOSettings^.ud_AddressRd := DeviceAddress + DIASDRIVE_ADR_ALT_BUF_RD_OFFSET + i$UDINT*DIASDRIVE_OFFSET_AxisRead;
        newIsoDOs[i].p_DOSettings^.ud_AddressWr := DeviceAddress + DIASDRIVE_ADR_ALT_BUF_WR_OFFSET + i$UDINT*DIASDRIVE_OFFSET_AxisRead;
      end_if;
      //set right para state
      aAxisData[i].us_ParaReady := _IdleState;
      aAxisData[i].e_AxisState := _NoInit;
    end_for;

    if TempFetchDigitalInputs then
      if b_PayloadSupport then
        if bAddDOsToListSupport then
          sd_retval := MULTI_VARAN_IINSERTDOINTODOL(newDigInDO.p_Handle$UDINT);
        end_if;
        EnableDO(ud_DOHandle:=newDigInDO.p_Handle$UDINT);
      else
      newDigInDO.p_DOSettings^.ud_Address := DeviceAddress + DIASDRIVE_ADR_INPUTS;

      // start getting the inputs
      ResetDataObject	( p_handleDO	:= newDigInDO.p_Handle
                      , us_state		:= VARAN_DO_CONT_RUN
                      , ud_bytes		:= sizeof(USINT)
                      );
      end_if;
    end_if;
    b_AlreadyConnected := TRUE;
  end_if;

END_FUNCTION

FUNCTION _VaranDriveBase::InstallDefaultDO
VAR
  sd_retval : DINT;
  tmp_dol_type : UDINT;
END_VAR

  if (CreatedCompDOs = FALSE) then
    //-----------------------------------------------------------------------------------------------
    //install default data object for the first axis

    //set right data object length
    if ExtendedAxisSettings AND 1 then
      aAxisData[0].ud_DOLength := sizeof(t_DataReadOneAxis);
      aAxisData[0].b_ExtendedAxis := TRUE;
    else
      aAxisData[0].ud_DOLength := sizeof(t_DataReadOneAxis) - 3 * sizeof(DINT);
      aAxisData[0].b_ExtendedAxis := FALSE;
    end_if;

    // check for fastaxis
    if FastAxisSettings AND 1 then
      aAxisData[0].b_FastAxis := TRUE;
    else
      aAxisData[0].b_FastAxis := FALSE;
    end_if;

    //install data object
    if b_PayloadSupport then
      tmp_dol_type := VARAN_DOL_ISO;

      if bAddDOsToListSupport then
        tmp_dol_Type := tmp_dol_Type OR VARAN_DOL_NOT_INSERT_DO_INTO_DOL;
      end_if;

      sd_retval := AddRdWrPayloadDO(  ud_dol_type     := tmp_dol_type
                                    , p_ud_handle     := ( #aDataObjects[0].p_Handle )$^UDINT
                                    , ud_offset_read  := DIASDRIVE_OFFSET_AxisRead
                                    , ud_length_read  := aAxisData[0].ud_DOLength
                                    , p_ud_data_read  := ( #aDataObjects[0].p_DataRead )$^UDINT
                                    , ud_offset_write := 0
                                    , ud_length_write := aAxisData[0].ud_DOLength
                                    , p_ud_data_write := ( #aDataObjects[0].p_DataWrite )$^UDINT
                                    , ud_type         := VM_MEMORY_ACCESS);

      //look if an error occurs
      if ( sd_retval <> VARANMANAGER_OK ) then
        State := _CreateDOFailed;
        return;
      end_if;
    else
    sd_retval := VaranIn.AddRdWrDO	( p_us_position_info:= p_VaranPosition
                    , ud_dol_type		:= VARAN_DOL_ISO
                    , p_ud_handle		:= ( #aDataObjects[0].p_Handle )$^UDINT
                    , ud_address_read	:= 0
                    , ud_length_read	:= aAxisData[0].ud_DOLength
                    , p_ud_data_read	:= ( #aDataObjects[0].p_DataRead )$^UDINT
                    , ud_address_write	:= 0
                    , ud_length_write	:= aAxisData[0].ud_DOLength
                    , p_ud_data_write	:= ( #aDataObjects[0].p_DataWrite )$^UDINT
                    , ud_type			:= VM_MEMORY_ACCESS
                    );

      //look if an error occurs
      if ( sd_retval <> VARANMANAGER_OK ) then
        State := _CreateDOFailed;
        return;
      end_if;
    end_if;

    //get address pointer to change address later when module is connected
    aDataObjects[0].p_DOSettings := (aDataObjects[0].p_DataWrite)$^t_VaranDOSettingsRdWr - VM_DO_OFFSET_RDWR;

    CreatedCompDOs := TRUE;
  end_if;

  if (b_AlreadyConnected = FALSE) & CreatedCompDOs then
    b_AlreadyConnected := TRUE;
    if b_PayloadSupport =FALSE then
    //correct address for data object read/write Axis 1
    aDataObjects[0].p_DOSettings^.ud_AddressRd := DeviceAddress + DIASDRIVE_OFFSET_AxisRead;
    aDataObjects[0].p_DOSettings^.ud_AddressWr := DeviceAddress;
    end_if;

    //set enable outputs in DCB
    //with VAC012 the hardware enables the outputs
    if ( DeviceID = VAC011_DEVICE_ID ) then
      aDataObjects[0].p_DataWrite^.us_DriveControl := 2#00111000;
    end_if;

    //set transmit register
    if aAxisData[0].b_ExtendedAxis then
      aDataObjects[0].p_DataWrite^.us_TransmitExecution.EnableValue3_5 := TRUE;
    end_if;

    //set right para state
    aAxisData[0].us_ParaReady := _IdleState;
    aAxisData[0].e_AxisState := _NoInit;
  end_if;

END_FUNCTION
